RoboDK station: Stringer A - Top Up - BOX1.rdk

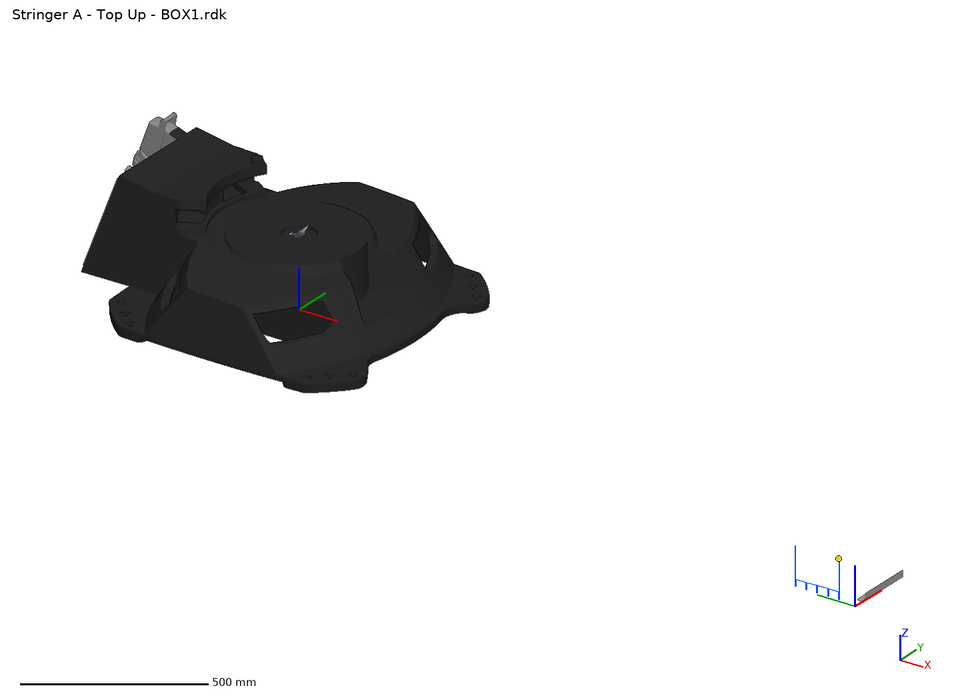
[picture v0: the station drawn from its stored meshes, robots at their saved joint values, targets as dots, program paths as lines]
Station Stringer A - Top Up - BOX1 (saved by RoboDK 5.2.3). Poses are relative to the parent item; angles as X-Y-Z fixed-axis rotations.
  - frame KUKA KR 210 R2700 extra Base at (0, 0, 0) mm
    - robot KUKA KR 210 R2700 extra: 6 axes, payload 210 kg, reach 2696 mm, repeatability 0.06 mm, weight 1068 kg
        joint limits [-185, -140, -120, -350, -125, -350] to [185, -5, 155, 350, 125, 350]; home [0, -90, 90, 0, 0, 0]; saved at [-7.543, -28.204, 108.426, 170.291, 29.33, -177.391]
      - tool Spindle, TCP at (32, 0, 260) mm, rotated rx 0 ry 39 rz 0 deg, size 157.3 x 72 x 259.9 mm
  - frame Frame 2 at (1800, 0, -372.68) mm, rotated rx 0 ry 0 rz 90 deg
    - object Stringer A-TopUP-BOX1 at (0, 22.5, 0) mm, rotated rx 0 ry 0 rz -90 deg, 5 curves, geometry from Point 5
    - object L-Stringer A - top up at (0, 0, 0) mm, size 183.1 x 20 x 20 mm, geometry from L-Stringer A - top up.stl
  - machining project Point settings: rotZ(0) | rotX(0)*rotY(0) | rotz(0) | onStart | onPathStart | onApproach | onPoint | onRetract | onFinish | SetRPM(%1) | SetTool(%1) | Extruder(%1) | default | default | OutOnMov(%1) | OutOffMov(%1) | onPathFinish | M_RunCode(%1)
  - program Point (36 instructions, listed below)
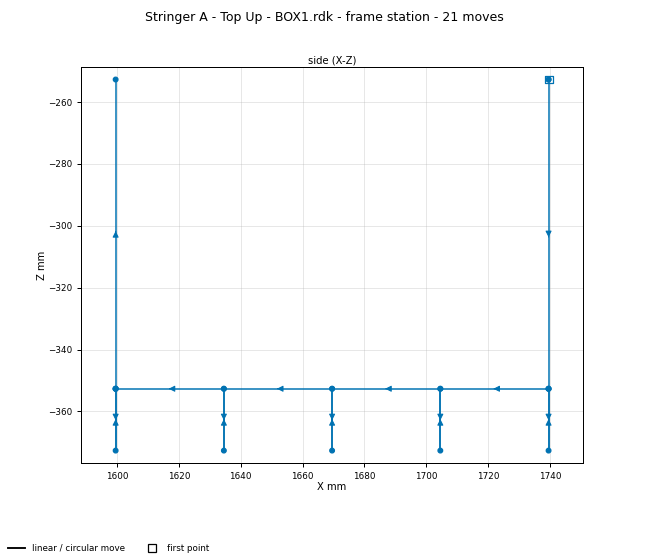
[picture p0: tool path of Stringer A - Top Up - BOX1.rdk in frame station, 21 of 21 moves have a stored position in this frame; points joined in program order, loops and branches not executed]

--- program Point (robot KUKA KR 210 R2700 extra) ---
  Smooth(1)
  Set speed (1000.0 mm/s)
  Set Ref.: Frame 2
  Set Tool: Spindle
  Show Spindle
  MoveJ 1 to (10.2, 60.43, 120) mm, rotated rx 180 ry 0 rz 180 deg; joints [-2.286, -34.025, 111.911, 176.819, 26.9, -178.94]
  MoveL 2 to (10.2, 60.43, 120) mm, rotated rx 180 ry 0 rz 180 deg; joints [-2.286, -34.025, 111.911, 176.819, 26.9, -178.94]
  MoveL 3 to (10.2, 60.43, 20) mm, rotated rx -180 ry 0 rz -180 deg; joints [-2.286, -28.692, 109.267, 177.085, 29.585, -179.242]
  MoveL 4 to (10.2, 60.43, 20) mm, rotated rx -180 ry 0 rz -180 deg; joints [-2.286, -28.692, 109.267, 177.085, 29.585, -179.242]
  Set speed (50.0 mm/s)
  MoveL 5 to (10.2, 60.43, 0) mm, rotated rx -180 ry 0 rz -180 deg; joints [-2.286, -27.634, 108.691, 177.128, 30.067, -179.291]
  MoveL 6 to (10.2, 60.43, 20) mm, rotated rx -180 ry 0 rz -180 deg; joints [-2.286, -28.692, 109.267, 177.085, 29.585, -179.242]
  Set speed (1000.0 mm/s)
  MoveL 7 to (10.2, 95.43, 20) mm, rotated rx 180 ry 0 rz -180 deg; joints [-3.608, -28.679, 109.174, 175.39, 29.519, -178.792]
  Set speed (50.0 mm/s)
  MoveL 8 to (10.2, 95.43, 0) mm, rotated rx -180 ry 0 rz -180 deg; joints [-3.608, -27.622, 108.598, 175.457, 29.999, -178.869]
  MoveL 9 to (10.2, 95.43, 20) mm, rotated rx 180 ry 0 rz -180 deg; joints [-3.608, -28.679, 109.174, 175.39, 29.519, -178.792]
  Set speed (1000.0 mm/s)
  MoveL 10 to (10.2, 130.43, 20) mm, rotated rx 180 ry 0 rz 180 deg; joints [-4.925, -28.661, 109.039, 173.686, 29.423, -178.326]
  Set speed (50.0 mm/s)
  MoveL 11 to (10.2, 130.43, 0) mm, rotated rx 180 ry 0 rz 180 deg; joints [-4.925, -27.605, 108.464, 173.778, 29.901, -178.432]
  MoveL 12 to (10.2, 130.43, 20) mm, rotated rx 180 ry 0 rz 180 deg; joints [-4.925, -28.661, 109.039, 173.686, 29.423, -178.326]
  Set speed (1000.0 mm/s)
  MoveL 13 to (10.2, 165.43, 20) mm, rotated rx 180 ry 0 rz 180 deg; joints [-6.237, -28.637, 108.862, 171.969, 29.299, -177.84]
  Set speed (50.0 mm/s)
  MoveL 14 to (10.2, 165.43, 0) mm, rotated rx -180 ry 0 rz -180 deg; joints [-6.237, -27.582, 108.287, 172.086, 29.775, -177.975]
  MoveL 15 to (10.2, 165.43, 20) mm, rotated rx 180 ry 0 rz 180 deg; joints [-6.237, -28.637, 108.862, 171.969, 29.299, -177.84]
  Set speed (1000.0 mm/s)
  MoveL 16 to (10.2, 200.43, 20) mm, rotated rx -180 ry 0 rz -180 deg; joints [-7.543, -28.606, 108.643, 170.235, 29.148, -177.327]
  Set speed (50.0 mm/s)
  MoveL 17 to (10.2, 200.43, 0) mm, rotated rx -180 ry 0 rz -180 deg; joints [-7.543, -27.553, 108.069, 170.378, 29.62, -177.492]
  MoveL 18 to (10.2, 200.43, 20) mm, rotated rx -180 ry 0 rz -180 deg; joints [-7.543, -28.606, 108.643, 170.235, 29.148, -177.327]
  MoveL 19 to (10.2, 200.43, 20) mm, rotated rx -180 ry 0 rz -180 deg; joints [-7.543, -28.606, 108.643, 170.235, 29.148, -177.327]
  Set speed (1000.0 mm/s)
  MoveL 20 to (10.2, 200.43, 20) mm, rotated rx -180 ry 0 rz -180 deg; joints [-7.543, -28.606, 108.643, 170.235, 29.148, -177.327]
  MoveL 21 to (10.2, 200.43, 120) mm, rotated rx 180 ry 0 rz -180 deg; joints [-7.543, -33.907, 111.275, 169.339, 26.521, -176.314]
